ABB RAPID module: Module_RDS.mod

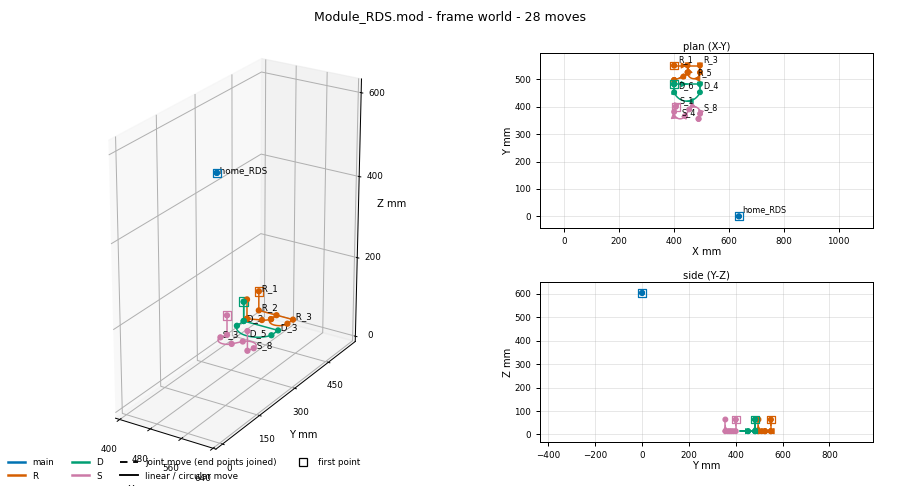
[picture p0: tool path of Module_RDS.mod in frame world, 28 of 28 moves have a stored position in this frame; points joined in program order, loops and branches not executed]
MODULE Module_RDS
    CONST robtarget home_RDS:=[[636.195461814,0,604.5],[0.5,0,0.866025404,0],[0,0,0,0],[9E+09,9E+09,9E+09,9E+09,9E+09,9E+09]];
    CONST robtarget R_1:=[[0,0,50],[0,0,1,0],[0,0,1,0],[9E+09,9E+09,9E+09,9E+09,9E+09,9E+09]];
    CONST robtarget R_2:=[[0,0,0],[0,0,1,0],[0,0,1,0],[9E+09,9E+09,9E+09,9E+09,9E+09,9E+09]];
    CONST robtarget R_3:=[[0,94,0],[0,0,1,0],[0,0,1,0],[9E+09,9E+09,9E+09,9E+09,9E+09,9E+09]];
    CONST robtarget R_4:=[[25.5,94,0],[0,0,1,0],[0,0,1,0],[9E+09,9E+09,9E+09,9E+09,9E+09,9E+09]];
    CONST robtarget R_5:=[[48,71.5,0],[0,0,1,0],[0,0,1,0],[9E+09,9E+09,9E+09,9E+09,9E+09,9E+09]];
    CONST robtarget R_6:=[[25,49,0],[0,0,1,0],[0,0,1,0],[9E+09,9E+09,9E+09,9E+09,9E+09,9E+09]];
    CONST robtarget R_7:=[[0,49,0],[0,0,1,0],[0,0,1,0],[9E+09,9E+09,9E+09,9E+09,9E+09,9E+09]];
    CONST robtarget R_8:=[[34.5,43,0],[0,0,1,0],[0,0,1,0],[9E+09,9E+09,9E+09,9E+09,9E+09,9E+09]];
    CONST robtarget R_9:=[[40.5,33.5,0],[0,0,1,0],[0,0,0,0],[9E+09,9E+09,9E+09,9E+09,9E+09,9E+09]];
    CONST robtarget R_10:=[[53,0,0],[0,0,1,0],[0,0,0,0],[9E+09,9E+09,9E+09,9E+09,9E+09,9E+09]];
    CONST robtarget R_11:=[[53,0,0],[0,0,1,0],[0,0,0,0],[9E+09,9E+09,9E+09,9E+09,9E+09,9E+09]];
    CONST robtarget D_1:=[[67.6,0,50],[0,0,1,0],[0,0,0,0],[9E+09,9E+09,9E+09,9E+09,9E+09,9E+09]];
    CONST robtarget D_2:=[[67.6,0,0],[0,0,1,0],[0,0,1,0],[9E+09,9E+09,9E+09,9E+09,9E+09,9E+09]];
    CONST robtarget D_3:=[[67.6,94,0],[0,0,1,0],[0,0,1,0],[9E+09,9E+09,9E+09,9E+09,9E+09,9E+09]];
    CONST robtarget D_4:=[[97.5,94,0],[0,0,1,0],[0,0,1,0],[9E+09,9E+09,9E+09,9E+09,9E+09,9E+09]];
    CONST robtarget D_5:=[[130,47,0],[0,0,1,0],[0,0,1,0],[9E+09,9E+09,9E+09,9E+09,9E+09,9E+09]];
    CONST robtarget D_6:=[[97.5,0,0],[0,0,1,0],[0,0,1,0],[9E+09,9E+09,9E+09,9E+09,9E+09,9E+09]];
    CONST robtarget R_12:=[[53,0,50],[0,0,1,0],[0,0,1,0],[9E+09,9E+09,9E+09,9E+09,9E+09,9E+09]];
    CONST robtarget S_1:=[[150,6,50],[0,0,1,0],[0,0,0,0],[9E+09,9E+09,9E+09,9E+09,9E+09,9E+09]];
    CONST robtarget S_2:=[[150,6,0],[0,0,1,0],[0,0,1,0],[9E+09,9E+09,9E+09,9E+09,9E+09,9E+09]];
    CONST robtarget S_3:=[[169,0,0],[0,0,1,0],[0,0,1,0],[9E+09,9E+09,9E+09,9E+09,9E+09,9E+09]];
    CONST robtarget S_4:=[[193,14,0],[0,0,1,0],[0,0,1,0],[9E+09,9E+09,9E+09,9E+09,9E+09,9E+09]];
    CONST robtarget S_5:=[[184,40,0],[0,0,1,0],[0,0,1,0],[9E+09,9E+09,9E+09,9E+09,9E+09,9E+09]];
    CONST robtarget S_6:=[[160,55,0],[0,0,1,0],[0,0,1,0],[9E+09,9E+09,9E+09,9E+09,9E+09,9E+09]];
    CONST robtarget S_7:=[[152,81,0],[0,0,1,0],[0,0,1,0],[9E+09,9E+09,9E+09,9E+09,9E+09,9E+09]];
    CONST robtarget S_8:=[[176,94.5,0],[0,0,1,0],[0,0,1,0],[9E+09,9E+09,9E+09,9E+09,9E+09,9E+09]];
    CONST robtarget S_9:=[[194.5,89,0],[0,0,1,0],[0,0,0,0],[9E+09,9E+09,9E+09,9E+09,9E+09,9E+09]];
    CONST robtarget S_10:=[[194.5,89,50],[0,0,1,0],[0,0,0,0],[9E+09,9E+09,9E+09,9E+09,9E+09,9E+09]];
    CONST robtarget R_1_2:=[[0,0,50],[0,0,1,0],[-1,1,-1,0],[9E+09,9E+09,9E+09,9E+09,9E+09,9E+09]];
    CONST robtarget R_2_2:=[[0,0,0],[0,0,1,0],[-1,1,-1,0],[9E+09,9E+09,9E+09,9E+09,9E+09,9E+09]];
    CONST robtarget R_3_2:=[[0,94,0],[0,0,1,0],[-1,0,0,0],[9E+09,9E+09,9E+09,9E+09,9E+09,9E+09]];
    CONST robtarget R_4_2:=[[25.5,94,0],[0,0,1,0],[-1,0,0,0],[9E+09,9E+09,9E+09,9E+09,9E+09,9E+09]];
    CONST robtarget R_5_2:=[[48,71.5,0],[0,0,1,0],[-1,0,0,0],[9E+09,9E+09,9E+09,9E+09,9E+09,9E+09]];
    CONST robtarget R_6_2:=[[25,49,0],[0,0,1,0],[-1,1,-1,0],[9E+09,9E+09,9E+09,9E+09,9E+09,9E+09]];
    CONST robtarget R_7_2:=[[0,49,0],[0,0,1,0],[-1,1,-1,0],[9E+09,9E+09,9E+09,9E+09,9E+09,9E+09]];
    CONST robtarget R_8_2:=[[34.5,43,0],[0,0,1,0],[-1,1,-1,0],[9E+09,9E+09,9E+09,9E+09,9E+09,9E+09]];
    CONST robtarget R_9_2:=[[40.5,33.5,0],[0,0,1,0],[-1,1,-1,0],[9E+09,9E+09,9E+09,9E+09,9E+09,9E+09]];
    CONST robtarget R_10_2:=[[53,0,0],[0,0,1,0],[-1,1,-1,0],[9E+09,9E+09,9E+09,9E+09,9E+09,9E+09]];
    CONST robtarget R_11_2:=[[53,0,0],[0,0,1,0],[-1,1,-1,0],[9E+09,9E+09,9E+09,9E+09,9E+09,9E+09]];
    CONST robtarget R_12_2:=[[53,0,50],[0,0,1,0],[-1,1,-1,0],[9E+09,9E+09,9E+09,9E+09,9E+09,9E+09]];
    CONST robtarget D_1_2:=[[67.6,0,50],[0,0,1,0],[0,0,0,0],[9E+09,9E+09,9E+09,9E+09,9E+09,9E+09]];
    CONST robtarget D_2_2:=[[67.6,0,0],[0,0,1,0],[-1,1,-1,0],[9E+09,9E+09,9E+09,9E+09,9E+09,9E+09]];
    CONST robtarget D_3_2:=[[67.6,94,0],[0,0,1,0],[-1,0,0,0],[9E+09,9E+09,9E+09,9E+09,9E+09,9E+09]];
    CONST robtarget D_4_2:=[[97.5,94,0],[0,0,1,0],[-1,0,0,0],[9E+09,9E+09,9E+09,9E+09,9E+09,9E+09]];
    CONST robtarget D_5_2:=[[130,47,0],[0,0,1,0],[-1,0,-1,0],[9E+09,9E+09,9E+09,9E+09,9E+09,9E+09]];
    CONST robtarget D_6_2:=[[97.5,0,0],[0,0,1,0],[-1,1,-1,0],[9E+09,9E+09,9E+09,9E+09,9E+09,9E+09]];
    CONST robtarget S_1_2:=[[150,6,50],[0,0,1,0],[0,0,0,0],[9E+09,9E+09,9E+09,9E+09,9E+09,9E+09]];
    CONST robtarget S_2_2:=[[150,6,0],[0,0,1,0],[-1,0,-1,0],[9E+09,9E+09,9E+09,9E+09,9E+09,9E+09]];
    CONST robtarget S_3_2:=[[169,0,0],[0,0,1,0],[-1,0,-1,0],[9E+09,9E+09,9E+09,9E+09,9E+09,9E+09]];
    CONST robtarget S_4_2:=[[193,14,0],[0,0,1,0],[-1,0,-1,0],[9E+09,9E+09,9E+09,9E+09,9E+09,9E+09]];
    CONST robtarget S_5_2:=[[184,40,0],[0,0,1,0],[-1,0,-1,0],[9E+09,9E+09,9E+09,9E+09,9E+09,9E+09]];
    CONST robtarget S_6_2:=[[160,55,0],[0,0,1,0],[-1,0,-1,0],[9E+09,9E+09,9E+09,9E+09,9E+09,9E+09]];
    CONST robtarget S_7_2:=[[152,81,0],[0,0,1,0],[-1,0,0,0],[9E+09,9E+09,9E+09,9E+09,9E+09,9E+09]];
    CONST robtarget S_8_2:=[[176,94.5,0],[0,0,1,0],[-1,0,0,0],[9E+09,9E+09,9E+09,9E+09,9E+09,9E+09]];
    CONST robtarget S_9_2:=[[194.5,89,0],[0,0,1,0],[-1,0,0,0],[9E+09,9E+09,9E+09,9E+09,9E+09,9E+09]];
    CONST robtarget S_10_2:=[[194.5,89,50],[0,0,1,0],[-1,0,0,0],[9E+09,9E+09,9E+09,9E+09,9E+09,9E+09]];
    PERS tooldata TCP_Porta_marcador:=[TRUE,[[0,0,150],[1,0,0,0]],[1,[0,0,1],[1,0,0,0],0,0,0]];
    TASK PERS wobjdata Workobject_1:=[FALSE,TRUE,"",[[0,0,0],[1,0,0,0]],[[400,550,14],[0.707106781,0,0,-0.707106781]]];
!***********************************************************
    !
    ! Módulo:  Module1
    !
    ! Descripción:
    !   <Introduzca la descripción aquí>
    !
    ! Autor: difao
    !
    ! Versión: 1.0
    !
    !***********************************************************


    !***********************************************************
    !
    ! Procedimiento Main
    !
    !   Este es el punto de entrada de su programa
    !
    !***********************************************************
    PROC main()
        !Añada aquí su código
        MoveJ home_RDS,v200,fine,TCP_Porta_marcador\WObj:=wobj0;
        R;
        D;
        S;
        MoveJ home_RDS,v200,fine,TCP_Porta_marcador\WObj:=wobj0;
    ENDPROC
    PROC R()
        MoveJ R_1,v200,fine,TCP_Porta_marcador\WObj:=Workobject_1;
        MoveL R_2,v100,fine,TCP_Porta_marcador\WObj:=Workobject_1;
        MoveL R_3,v100,fine,TCP_Porta_marcador\WObj:=Workobject_1;
        MoveL R_4,v100,fine,TCP_Porta_marcador\WObj:=Workobject_1;
        MoveC R_5,R_6,v100,fine,TCP_Porta_marcador\WObj:=Workobject_1;
        MoveL R_7,v100,fine,TCP_Porta_marcador\WObj:=Workobject_1;
        MoveL R_6,v100,fine,TCP_Porta_marcador\WObj:=Workobject_1;
        MoveC R_8,R_9,v100,fine,TCP_Porta_marcador\WObj:=Workobject_1;
        MoveL R_10,v100,fine,TCP_Porta_marcador\WObj:=Workobject_1;
        MoveL R_11,v100,fine,TCP_Porta_marcador\WObj:=Workobject_1;
        MoveL R_12,v100,fine,TCP_Porta_marcador\WObj:=Workobject_1;
    ENDPROC
    PROC D()
        MoveL D_1,v100,fine,TCP_Porta_marcador\WObj:=Workobject_1;
        MoveL D_2,v100,fine,TCP_Porta_marcador\WObj:=Workobject_1;
        MoveL D_3,v100,fine,TCP_Porta_marcador\WObj:=Workobject_1;
        MoveL D_4,v100,fine,TCP_Porta_marcador\WObj:=Workobject_1;
        MoveC D_5,D_6,v100,fine,TCP_Porta_marcador\WObj:=Workobject_1;
        MoveL D_2,v100,fine,TCP_Porta_marcador\WObj:=Workobject_1;
        MoveL D_1,v100,fine,TCP_Porta_marcador\WObj:=Workobject_1;
    ENDPROC
    PROC S()
        MoveL S_1,v100,fine,TCP_Porta_marcador\WObj:=Workobject_1;
        MoveL S_2,v100,fine,TCP_Porta_marcador\WObj:=Workobject_1;
        MoveL S_3,v100,fine,TCP_Porta_marcador\WObj:=Workobject_1;
        MoveC S_4,S_5,v100,fine,TCP_Porta_marcador\WObj:=Workobject_1;
        MoveL S_6,v100,fine,TCP_Porta_marcador\WObj:=Workobject_1;
        MoveC S_7,S_8,v100,fine,TCP_Porta_marcador\WObj:=Workobject_1;
        MoveL S_9,v100,fine,TCP_Porta_marcador\WObj:=Workobject_1;
        MoveL S_10,v100,fine,TCP_Porta_marcador\WObj:=Workobject_1;
    ENDPROC
ENDMODULE
